// TIA Portal V15 export
// export: Created 2018-02-11T06:44:35.9692027Z, ExportSetting None, DisplayName Totally Integrated Automation Portal, DisplayVersion V15, DisplayName TIA Portal Openness, DisplayVersion V15, DisplayName TIA Portal Teamcenter Gateway, DisplayVersion V15, DisplayName SINAMICS Startdrive Advanced, DisplayVersion V15, DisplayName G110M, G120, G120C, G120D, G120P, DisplayVersion V15, DisplayName G130, G150, S120, S150, SINAMICS MV, DisplayVersion V15, DisplayName STEP 7 Professional, DisplayVersion V15, DisplayName WinCC Professional, DisplayVersion V15, DisplayName SIMATIC Visualization Architect, DisplayVersion V15
DATA_BLOCK "Workshop1_DB"   // DB3
{ S7_Optimized_Access := 'TRUE' }
// stored: InstanceOfName Workshop1
"Workshop1"
BEGIN
END_DATA_BLOCK
